TYPE ST_System_WP_Parameter :
STRUCT
	AutoQuittierung			: BOOL ;
END_STRUCT
END_TYPE

(* stored: Version 1.1.0.1, ProductVersion 3.1.4024.9
   DUT ST_System_WP_Parameter: Id {c5714c85-b0c6-42a5-898a-5a864d4bd630} *)
